(* IEC 61131-3 sources: Industry-PLC-LLM/data/PLCBEAD_repo/PLCBEAD_PLCEmbed-main/PLC-BEAD/Source/GEB/SCALE, 1 file *)

(* ---- SCALE.ST ---- *)
FUNCTION SCALE:REAL

	VAR_INPUT
		X :	REAL;
		K :	REAL;
		O :	REAL;
		MX :	REAL;
		MN :	REAL;
	END_VAR

	SCALE := LIMIT(MN, X * K + O, MX);

END_FUNCTION

PROGRAM program0
  VAR
    X :	REAL;
	K :	REAL;
	O :	REAL;
	MX :	REAL;
	MN :	REAL;
    CEIL5_OUT : REAL;
  END_VAR

  CEIL5_OUT := SCALE(X, K, O, MX, MN);
END_PROGRAM
